KUKA KRL program: DEMO_MULTIPROC03.src, DEMO_MULTIPROC03.dat

--- DEMO_MULTIPROC03.src ---
&ACCESS RVO
&REL 23
&COMMENT MultiProc03
&PARAM DISKPATH = KRC:\R1\Program\PlcDemo
DEF  DEMO_MULTIPROC03 ( )
;********************************

;CREATOR : SPEEDBOT
;DATE    : 2024-09-23
;PROGRAM : DEMO_MULTIPROC03

;********************************
;FOLD INI;%{PE}
  ;FOLD BASISTECH INI
    GLOBAL INTERRUPT DECL 3 WHEN $STOPMESS==TRUE DO IR_STOPM ( )
    INTERRUPT ON 3
    BAS (#INITMOV,0 )
  ;ENDFOLD (BASISTECH INI)
  ;FOLD USER INI
    ;Make your modifications here
    continue
    if $MOVE_BCO == FALSE Then
      ; BCO
      ptp cur_jpos_()
    endif
  ;ENDFOLD (USER INI)
;ENDFOLD (INI)

;Example program for Process 1

;waiting for PLC clearance to proceed
;FOLD PLC.RequestToContinue ;%{PE}
req_to_continue_()
;ENDFOLD
;FOLD PLC.PathSegment IN Segment Nr: 124 ;%{PE}
path_segment_(124)
;ENDFOLD

;entering interference zone 1 with robot *.
;Enter Zone With R***
;FOLD PLC.EnterZone IN Zone Nr: ZONE [1] ;%{PE}
zone_ctrl_(#I_ENTER, 1)
;ENDFOLD

;Teach the robot to execute the first process trajectory.
;FOLD SPTP P1 CONT Vel=100 % PDAT1 Tool[1] Base[0] ;%{PE}
;FOLD Parameters ;%{h}
;Params IlfProvider=kukaroboter.basistech.inlineforms.movement.spline; Kuka.IsGlobalPoint=False; Kuka.PointName=P1; Kuka.BlendingEnabled=True; Kuka.MoveDataPtpName=PDAT1; Kuka.VelocityPtp=100; Kuka.VelocityFieldEnabled=True; Kuka.ColDetectFieldEnabled=True; Kuka.CurrentCDSetIndex=0; Kuka.MovementParameterFieldEnabled=True; IlfCommand=SPTP
;ENDFOLD
SPTP XP1 WITH $VEL_AXIS[1] = SVEL_JOINT(100.0), $TOOL = STOOL2(FP1), $BASE = SBASE(FP1.BASE_NO), $IPO_MODE = SIPO_MODE(FP1.IPO_FRAME), $LOAD = SLOAD(FP1.TOOL_NO), $ACC_AXIS[1] = SACC_JOINT(PPDAT1), $APO = SAPO_PTP(PPDAT1), $GEAR_JERK[1] = SGEAR_JERK(PPDAT1), $COLLMON_TOL_PRO[1] = USE_CM_PRO_VALUES(0) C_Spl
;ENDFOLD
;FOLD SPTP P2 CONT Vel=100 % PDAT2 Tool[1] Base[0] ;%{PE}
;FOLD Parameters ;%{h}
;Params IlfProvider=kukaroboter.basistech.inlineforms.movement.spline; Kuka.IsGlobalPoint=False; Kuka.PointName=P2; Kuka.BlendingEnabled=True; Kuka.MoveDataPtpName=PDAT2; Kuka.VelocityPtp=100; Kuka.VelocityFieldEnabled=True; Kuka.ColDetectFieldEnabled=True; Kuka.CurrentCDSetIndex=0; Kuka.MovementParameterFieldEnabled=True; IlfCommand=SPTP
;ENDFOLD
SPTP XP2 WITH $VEL_AXIS[1] = SVEL_JOINT(100.0), $TOOL = STOOL2(FP2), $BASE = SBASE(FP2.BASE_NO), $IPO_MODE = SIPO_MODE(FP2.IPO_FRAME), $LOAD = SLOAD(FP2.TOOL_NO), $ACC_AXIS[1] = SACC_JOINT(PPDAT2), $APO = SAPO_PTP(PPDAT2), $GEAR_JERK[1] = SGEAR_JERK(PPDAT2), $COLLMON_TOL_PRO[1] = USE_CM_PRO_VALUES(0) C_Spl
;ENDFOLD
;FOLD SPTP P3 CONT Vel=100 % PDAT3 Tool[1] Base[0] ;%{PE}
;FOLD Parameters ;%{h}
;Params IlfProvider=kukaroboter.basistech.inlineforms.movement.spline; Kuka.IsGlobalPoint=False; Kuka.PointName=P3; Kuka.BlendingEnabled=True; Kuka.MoveDataPtpName=PDAT3; Kuka.VelocityPtp=100; Kuka.VelocityFieldEnabled=True; Kuka.ColDetectFieldEnabled=True; Kuka.CurrentCDSetIndex=0; Kuka.MovementParameterFieldEnabled=True; IlfCommand=SPTP
;ENDFOLD
SPTP XP3 WITH $VEL_AXIS[1] = SVEL_JOINT(100.0), $TOOL = STOOL2(FP3), $BASE = SBASE(FP3.BASE_NO), $IPO_MODE = SIPO_MODE(FP3.IPO_FRAME), $LOAD = SLOAD(FP3.TOOL_NO), $ACC_AXIS[1] = SACC_JOINT(PPDAT3), $APO = SAPO_PTP(PPDAT3), $GEAR_JERK[1] = SGEAR_JERK(PPDAT3), $COLLMON_TOL_PRO[1] = USE_CM_PRO_VALUES(0) C_Spl
;ENDFOLD
;FOLD SLIN P4 CONT Vel=2 m/s CPDAT1 Tool[1] Base[0] ;%{PE}
;FOLD Parameters ;%{h}
;Params IlfProvider=kukaroboter.basistech.inlineforms.movement.spline; Kuka.IsGlobalPoint=False; Kuka.PointName=P4; Kuka.BlendingEnabled=True; Kuka.MoveDataName=CPDAT1; Kuka.VelocityPath=2; Kuka.VelocityFieldEnabled=True; Kuka.ColDetectFieldEnabled=True; Kuka.CurrentCDSetIndex=0; Kuka.MovementParameterFieldEnabled=True; IlfCommand=SLIN
;ENDFOLD
SLIN XP4 WITH $VEL = SVEL_CP(2.0, , LCPDAT1), $TOOL = STOOL2(FP4), $BASE = SBASE(FP4.BASE_NO), $IPO_MODE = SIPO_MODE(FP4.IPO_FRAME), $LOAD = SLOAD(FP4.TOOL_NO), $ACC = SACC_CP(LCPDAT1), $ORI_TYPE = SORI_TYP(LCPDAT1), $APO = SAPO(LCPDAT1), $JERK = SJERK(LCPDAT1), $COLLMON_TOL_PRO[1] = USE_CM_PRO_VALUES(0) C_Spl
;ENDFOLD
;FOLD SLIN P5 CONT Vel=2 m/s CPDAT2 Tool[1] Base[0] ;%{PE}
;FOLD Parameters ;%{h}
;Params IlfProvider=kukaroboter.basistech.inlineforms.movement.spline; Kuka.IsGlobalPoint=False; Kuka.PointName=P5; Kuka.BlendingEnabled=True; Kuka.MoveDataName=CPDAT2; Kuka.VelocityPath=2; Kuka.VelocityFieldEnabled=True; Kuka.ColDetectFieldEnabled=True; Kuka.CurrentCDSetIndex=0; Kuka.MovementParameterFieldEnabled=True; IlfCommand=SLIN
;ENDFOLD
SLIN XP5 WITH $VEL = SVEL_CP(2.0, , LCPDAT2), $TOOL = STOOL2(FP5), $BASE = SBASE(FP5.BASE_NO), $IPO_MODE = SIPO_MODE(FP5.IPO_FRAME), $LOAD = SLOAD(FP5.TOOL_NO), $ACC = SACC_CP(LCPDAT2), $ORI_TYPE = SORI_TYP(LCPDAT2), $APO = SAPO(LCPDAT2), $JERK = SJERK(LCPDAT2), $COLLMON_TOL_PRO[1] = USE_CM_PRO_VALUES(0) C_Spl
;ENDFOLD
;FOLD SLIN P6 CONT Vel=2 m/s CPDAT3 Tool[1] Base[0] ;%{PE}
;FOLD Parameters ;%{h}
;Params IlfProvider=kukaroboter.basistech.inlineforms.movement.spline; Kuka.IsGlobalPoint=False; Kuka.PointName=P6; Kuka.BlendingEnabled=True; Kuka.MoveDataName=CPDAT3; Kuka.VelocityPath=2; Kuka.VelocityFieldEnabled=True; Kuka.ColDetectFieldEnabled=True; Kuka.CurrentCDSetIndex=0; Kuka.MovementParameterFieldEnabled=True; IlfCommand=SLIN
;ENDFOLD
SLIN XP6 WITH $VEL = SVEL_CP(2.0, , LCPDAT3), $TOOL = STOOL2(FP6), $BASE = SBASE(FP6.BASE_NO), $IPO_MODE = SIPO_MODE(FP6.IPO_FRAME), $LOAD = SLOAD(FP6.TOOL_NO), $ACC = SACC_CP(LCPDAT3), $ORI_TYPE = SORI_TYP(LCPDAT3), $APO = SAPO(LCPDAT3), $JERK = SJERK(LCPDAT3), $COLLMON_TOL_PRO[1] = USE_CM_PRO_VALUES(0) C_Spl
;ENDFOLD
;FOLD SPTP P7 CONT Vel=100 % PDAT4 Tool[1] Base[0] ;%{PE}
;FOLD Parameters ;%{h}
;Params IlfProvider=kukaroboter.basistech.inlineforms.movement.spline; Kuka.IsGlobalPoint=False; Kuka.PointName=P7; Kuka.BlendingEnabled=True; Kuka.MoveDataPtpName=PDAT4; Kuka.VelocityPtp=100; Kuka.VelocityFieldEnabled=True; Kuka.ColDetectFieldEnabled=True; Kuka.CurrentCDSetIndex=0; Kuka.MovementParameterFieldEnabled=True; IlfCommand=SPTP
;ENDFOLD
SPTP XP7 WITH $VEL_AXIS[1] = SVEL_JOINT(100.0), $TOOL = STOOL2(FP7), $BASE = SBASE(FP7.BASE_NO), $IPO_MODE = SIPO_MODE(FP7.IPO_FRAME), $LOAD = SLOAD(FP7.TOOL_NO), $ACC_AXIS[1] = SACC_JOINT(PPDAT4), $APO = SAPO_PTP(PPDAT4), $GEAR_JERK[1] = SGEAR_JERK(PPDAT4), $COLLMON_TOL_PRO[1] = USE_CM_PRO_VALUES(0) C_Spl
;ENDFOLD
;FOLD SPTP P8 CONT Vel=100 % PDAT5 Tool[1] Base[0] ;%{PE}
;FOLD Parameters ;%{h}
;Params IlfProvider=kukaroboter.basistech.inlineforms.movement.spline; Kuka.IsGlobalPoint=False; Kuka.PointName=P8; Kuka.BlendingEnabled=True; Kuka.MoveDataPtpName=PDAT5; Kuka.VelocityPtp=100; Kuka.VelocityFieldEnabled=True; Kuka.ColDetectFieldEnabled=True; Kuka.CurrentCDSetIndex=0; Kuka.MovementParameterFieldEnabled=True; IlfCommand=SPTP
;ENDFOLD
SPTP XP8 WITH $VEL_AXIS[1] = SVEL_JOINT(100.0), $TOOL = STOOL2(FP8), $BASE = SBASE(FP8.BASE_NO), $IPO_MODE = SIPO_MODE(FP8.IPO_FRAME), $LOAD = SLOAD(FP8.TOOL_NO), $ACC_AXIS[1] = SACC_JOINT(PPDAT5), $APO = SAPO_PTP(PPDAT5), $GEAR_JERK[1] = SGEAR_JERK(PPDAT5), $COLLMON_TOL_PRO[1] = USE_CM_PRO_VALUES(0) C_Spl
;ENDFOLD

;This position has been fully cleared
;Does not interfere with the gripper and the corresponding robot.

;Report the completion of the first process cycle
;FOLD PLC.PathSegment IN Segment Nr: 154 ;%{PE}
path_segment_(154)
;ENDFOLD

;Exit the interference zone 1 with robot *.
;Enter Zone With R***
;FOLD PLC.ExitZone IN Zone Nr: ZONE [1] ;%{PE}
zone_ctrl_(#I_EXIT, 1)
;ENDFOLD

;waiting for PLC clearance to proceed
;FOLD PLC.RequestToContinue ;%{PE}
req_to_continue_()
;ENDFOLD
;FOLD PLC.PathSegment IN Segment Nr: 125 ;%{PE}
path_segment_(125)
;ENDFOLD

;entering interference zone 2 with robot *.
;Enter Zone With R***
;FOLD PLC.EnterZone IN Zone Nr: ZONE [2] ;%{PE}
zone_ctrl_(#I_ENTER, 2)
;ENDFOLD

;Teach the robot to execute the second process trajectory.
;FOLD SPTP P9 CONT Vel=100 % PDAT6 Tool[1] Base[0] ;%{PE}
;FOLD Parameters ;%{h}
;Params IlfProvider=kukaroboter.basistech.inlineforms.movement.spline; Kuka.IsGlobalPoint=False; Kuka.PointName=P9; Kuka.BlendingEnabled=True; Kuka.MoveDataPtpName=PDAT6; Kuka.VelocityPtp=100; Kuka.VelocityFieldEnabled=True; Kuka.ColDetectFieldEnabled=True; Kuka.CurrentCDSetIndex=0; Kuka.MovementParameterFieldEnabled=True; IlfCommand=SPTP
;ENDFOLD
SPTP XP9 WITH $VEL_AXIS[1] = SVEL_JOINT(100.0), $TOOL = STOOL2(FP9), $BASE = SBASE(FP9.BASE_NO), $IPO_MODE = SIPO_MODE(FP9.IPO_FRAME), $LOAD = SLOAD(FP9.TOOL_NO), $ACC_AXIS[1] = SACC_JOINT(PPDAT6), $APO = SAPO_PTP(PPDAT6), $GEAR_JERK[1] = SGEAR_JERK(PPDAT6), $COLLMON_TOL_PRO[1] = USE_CM_PRO_VALUES(0) C_Spl
;ENDFOLD
;FOLD SPTP P10 CONT Vel=100 % PDAT7 Tool[1] Base[0] ;%{PE}
;FOLD Parameters ;%{h}
;Params IlfProvider=kukaroboter.basistech.inlineforms.movement.spline; Kuka.IsGlobalPoint=False; Kuka.PointName=P10; Kuka.BlendingEnabled=True; Kuka.MoveDataPtpName=PDAT7; Kuka.VelocityPtp=100; Kuka.VelocityFieldEnabled=True; Kuka.ColDetectFieldEnabled=True; Kuka.CurrentCDSetIndex=0; Kuka.MovementParameterFieldEnabled=True; IlfCommand=SPTP
;ENDFOLD
SPTP XP10 WITH $VEL_AXIS[1] = SVEL_JOINT(100.0), $TOOL = STOOL2(FP10), $BASE = SBASE(FP10.BASE_NO), $IPO_MODE = SIPO_MODE(FP10.IPO_FRAME), $LOAD = SLOAD(FP10.TOOL_NO), $ACC_AXIS[1] = SACC_JOINT(PPDAT7), $APO = SAPO_PTP(PPDAT7), $GEAR_JERK[1] = SGEAR_JERK(PPDAT7), $COLLMON_TOL_PRO[1] = USE_CM_PRO_VALUES(0) C_Spl
;ENDFOLD
;FOLD SPTP P11 CONT Vel=100 % PDAT8 Tool[1] Base[0] ;%{PE}
;FOLD Parameters ;%{h}
;Params IlfProvider=kukaroboter.basistech.inlineforms.movement.spline; Kuka.IsGlobalPoint=False; Kuka.PointName=P11; Kuka.BlendingEnabled=True; Kuka.MoveDataPtpName=PDAT8; Kuka.VelocityPtp=100; Kuka.VelocityFieldEnabled=True; Kuka.ColDetectFieldEnabled=True; Kuka.CurrentCDSetIndex=0; Kuka.MovementParameterFieldEnabled=True; IlfCommand=SPTP
;ENDFOLD
SPTP XP11 WITH $VEL_AXIS[1] = SVEL_JOINT(100.0), $TOOL = STOOL2(FP11), $BASE = SBASE(FP11.BASE_NO), $IPO_MODE = SIPO_MODE(FP11.IPO_FRAME), $LOAD = SLOAD(FP11.TOOL_NO), $ACC_AXIS[1] = SACC_JOINT(PPDAT8), $APO = SAPO_PTP(PPDAT8), $GEAR_JERK[1] = SGEAR_JERK(PPDAT8), $COLLMON_TOL_PRO[1] = USE_CM_PRO_VALUES(0) C_Spl
;ENDFOLD
;FOLD SLIN P12 CONT Vel=2 m/s CPDAT4 Tool[1] Base[0] ;%{PE}
;FOLD Parameters ;%{h}
;Params IlfProvider=kukaroboter.basistech.inlineforms.movement.spline; Kuka.IsGlobalPoint=False; Kuka.PointName=P12; Kuka.BlendingEnabled=True; Kuka.MoveDataName=CPDAT4; Kuka.VelocityPath=2; Kuka.VelocityFieldEnabled=True; Kuka.ColDetectFieldEnabled=True; Kuka.CurrentCDSetIndex=0; Kuka.MovementParameterFieldEnabled=True; IlfCommand=SLIN
;ENDFOLD
SLIN XP12 WITH $VEL = SVEL_CP(2.0, , LCPDAT4), $TOOL = STOOL2(FP12), $BASE = SBASE(FP12.BASE_NO), $IPO_MODE = SIPO_MODE(FP12.IPO_FRAME), $LOAD = SLOAD(FP12.TOOL_NO), $ACC = SACC_CP(LCPDAT4), $ORI_TYPE = SORI_TYP(LCPDAT4), $APO = SAPO(LCPDAT4), $JERK = SJERK(LCPDAT4), $COLLMON_TOL_PRO[1] = USE_CM_PRO_VALUES(0) C_Spl
;ENDFOLD
;FOLD SLIN P13 CONT Vel=2 m/s CPDAT5 Tool[1] Base[0] ;%{PE}
;FOLD Parameters ;%{h}
;Params IlfProvider=kukaroboter.basistech.inlineforms.movement.spline; Kuka.IsGlobalPoint=False; Kuka.PointName=P13; Kuka.BlendingEnabled=True; Kuka.MoveDataName=CPDAT5; Kuka.VelocityPath=2; Kuka.VelocityFieldEnabled=True; Kuka.ColDetectFieldEnabled=True; Kuka.CurrentCDSetIndex=0; Kuka.MovementParameterFieldEnabled=True; IlfCommand=SLIN
;ENDFOLD
SLIN XP13 WITH $VEL = SVEL_CP(2.0, , LCPDAT5), $TOOL = STOOL2(FP13), $BASE = SBASE(FP13.BASE_NO), $IPO_MODE = SIPO_MODE(FP13.IPO_FRAME), $LOAD = SLOAD(FP13.TOOL_NO), $ACC = SACC_CP(LCPDAT5), $ORI_TYPE = SORI_TYP(LCPDAT5), $APO = SAPO(LCPDAT5), $JERK = SJERK(LCPDAT5), $COLLMON_TOL_PRO[1] = USE_CM_PRO_VALUES(0) C_Spl
;ENDFOLD
;FOLD SLIN P14 CONT Vel=2 m/s CPDAT6 Tool[1] Base[0] ;%{PE}
;FOLD Parameters ;%{h}
;Params IlfProvider=kukaroboter.basistech.inlineforms.movement.spline; Kuka.IsGlobalPoint=False; Kuka.PointName=P14; Kuka.BlendingEnabled=True; Kuka.MoveDataName=CPDAT6; Kuka.VelocityPath=2; Kuka.VelocityFieldEnabled=True; Kuka.ColDetectFieldEnabled=True; Kuka.CurrentCDSetIndex=0; Kuka.MovementParameterFieldEnabled=True; IlfCommand=SLIN
;ENDFOLD
SLIN XP14 WITH $VEL = SVEL_CP(2.0, , LCPDAT6), $TOOL = STOOL2(FP14), $BASE = SBASE(FP14.BASE_NO), $IPO_MODE = SIPO_MODE(FP14.IPO_FRAME), $LOAD = SLOAD(FP14.TOOL_NO), $ACC = SACC_CP(LCPDAT6), $ORI_TYPE = SORI_TYP(LCPDAT6), $APO = SAPO(LCPDAT6), $JERK = SJERK(LCPDAT6), $COLLMON_TOL_PRO[1] = USE_CM_PRO_VALUES(0) C_Spl
;ENDFOLD
;FOLD SPTP P15 CONT Vel=100 % PDAT9 Tool[1] Base[0] ;%{PE}
;FOLD Parameters ;%{h}
;Params IlfProvider=kukaroboter.basistech.inlineforms.movement.spline; Kuka.IsGlobalPoint=False; Kuka.PointName=P15; Kuka.BlendingEnabled=True; Kuka.MoveDataPtpName=PDAT9; Kuka.VelocityPtp=100; Kuka.VelocityFieldEnabled=True; Kuka.ColDetectFieldEnabled=True; Kuka.CurrentCDSetIndex=0; Kuka.MovementParameterFieldEnabled=True; IlfCommand=SPTP
;ENDFOLD
SPTP XP15 WITH $VEL_AXIS[1] = SVEL_JOINT(100.0), $TOOL = STOOL2(FP15), $BASE = SBASE(FP15.BASE_NO), $IPO_MODE = SIPO_MODE(FP15.IPO_FRAME), $LOAD = SLOAD(FP15.TOOL_NO), $ACC_AXIS[1] = SACC_JOINT(PPDAT9), $APO = SAPO_PTP(PPDAT9), $GEAR_JERK[1] = SGEAR_JERK(PPDAT9), $COLLMON_TOL_PRO[1] = USE_CM_PRO_VALUES(0) C_Spl
;ENDFOLD
;FOLD SPTP P16 CONT Vel=100 % PDAT10 Tool[1] Base[0] ;%{PE}
;FOLD Parameters ;%{h}
;Params IlfProvider=kukaroboter.basistech.inlineforms.movement.spline; Kuka.IsGlobalPoint=False; Kuka.PointName=P16; Kuka.BlendingEnabled=True; Kuka.MoveDataPtpName=PDAT10; Kuka.VelocityPtp=100; Kuka.VelocityFieldEnabled=True; Kuka.ColDetectFieldEnabled=True; Kuka.CurrentCDSetIndex=0; Kuka.MovementParameterFieldEnabled=True; IlfCommand=SPTP
;ENDFOLD
SPTP XP16 WITH $VEL_AXIS[1] = SVEL_JOINT(100.0), $TOOL = STOOL2(FP16), $BASE = SBASE(FP16.BASE_NO), $IPO_MODE = SIPO_MODE(FP16.IPO_FRAME), $LOAD = SLOAD(FP16.TOOL_NO), $ACC_AXIS[1] = SACC_JOINT(PPDAT10), $APO = SAPO_PTP(PPDAT10), $GEAR_JERK[1] = SGEAR_JERK(PPDAT10), $COLLMON_TOL_PRO[1] = USE_CM_PRO_VALUES(0) C_Spl
;ENDFOLD

;Report the completion of the second process cycle
;FOLD PLC.PathSegment IN Segment Nr: 155 ;%{PE}
path_segment_(155)
;ENDFOLD

;Exit the interference zone 2 with robot *.
;Enter Zone With R***
;FOLD PLC.ExitZone IN Zone Nr: ZONE [2] ;%{PE}
zone_ctrl_(#I_EXIT, 2)
;ENDFOLD
END

--- DEMO_MULTIPROC03.dat ---
&ACCESS RVO
&REL 23
&COMMENT MultiProc03
&PARAM DISKPATH = KRC:\R1\Program\PlcDemo
DEFDAT  DEMO_MULTIPROC03
;FOLD EXTERNAL DECLARATIONS;%{PE}%MKUKATPBASIS,%CEXT,%VCOMMON,%P
;FOLD BASISTECH EXT;%{PE}%MKUKATPBASIS,%CEXT,%VEXT,%P
EXT  BAS (BAS_COMMAND  :IN,REAL  :IN )
DECL INT SUCCESS
;ENDFOLD (BASISTECH EXT)
;FOLD USER EXT;%{E}%MKUKATPUSER,%CEXT,%VEXT,%P
;Make your modifications here

;ENDFOLD (USER EXT)
;ENDFOLD (EXTERNAL DECLARATIONS)
DECL E6POS XP1={X 0.00,Y 0.0,Z 0.00,A 0.0,B 0.0000,C 0.0,S 0,T 0,E1 0.0,E2 0.0,E3 0.0,E4 0.0,E5 0.0,E6 0.0}
DECL FDAT FP1={TOOL_NO 1,BASE_NO 0,IPO_FRAME #BASE,POINT2[] " "}
DECL PDAT PPDAT1={VEL 100.000,ACC 100.000,APO_DIST 500.000,APO_MODE #CDIS,GEAR_JERK 100.000,EXAX_IGN 0}
DECL MODULEPARAM_T LAST_TP_PARAMS={PARAMS[] "Kuka.VelocityFieldEnabled=True; Kuka.ColDetectFieldEnabled=True; Kuka.MovementParameterFieldEnabled=True; Kuka.IsAngleEnabled=False; Kuka.PointName=P8; Kuka.FrameData.base_no=0; Kuka.FrameData.tool_no=1; Kuka.FrameData.ipo_frame=#BASE; Kuka.isglobalpoint=False; Kuka.MoveDataPtpName=PDAT5; Kuka.MovementDataPdat.apo_mode=#CDIS; Kuka.MovementDataPdat.apo_dist=500; Kuka.MovementData.vel=100; Kuka.MovementData.acc=100; Kuka.MovementData.gear_jerk=100; Kuka.MovementData.exax_ign=0; Kuka.VelocityPtp=100; Kuka.BlendingEnabled=True; Kuka.CurrentCDSetIndex=0; Kuka.MoveDataName=CPDAT3; Kuka.MovementData.apo_fac=50; Kuka.MovementData.apo_dist=500; Kuka.MovementData.axis_acc=100; Kuka.MovementData.axis_vel=100; Kuka.MovementData.circ_typ=#BASE; Kuka.MovementData.jerk_fac=50; Kuka.MovementData.ori_typ=#VAR; Kuka.VelocityPath=2      "}
DECL E6POS XP2={X 0.00,Y 0.0,Z 0.00,A 0.0,B 0.0000,C 0.0,S 0,T 0,E1 0.0,E2 0.0,E3 0.0,E4 0.0,E5 0.0,E6 0.0}
DECL FDAT FP2={TOOL_NO 1,BASE_NO 0,IPO_FRAME #BASE,POINT2[] " "}
DECL PDAT PPDAT2={VEL 100.000,ACC 100.000,APO_DIST 500.000,APO_MODE #CDIS,GEAR_JERK 100.000,EXAX_IGN 0}
DECL E6POS XP3={X 0.00,Y 0.0,Z 0.00,A 0.0,B 0.0000,C 0.0,S 0,T 0,E1 0.0,E2 0.0,E3 0.0,E4 0.0,E5 0.0,E6 0.0}
DECL FDAT FP3={TOOL_NO 1,BASE_NO 0,IPO_FRAME #BASE,POINT2[] " "}
DECL PDAT PPDAT3={VEL 100.000,ACC 100.000,APO_DIST 500.000,APO_MODE #CDIS,GEAR_JERK 100.000,EXAX_IGN 0}
DECL E6POS XP4={X 0.00,Y 0.0,Z 0.00,A 0.0,B 0.0000,C 0.0,S 0,T 0,E1 0.0,E2 0.0,E3 0.0,E4 0.0,E5 0.0,E6 0.0}
DECL FDAT FP4={TOOL_NO 1,BASE_NO 0,IPO_FRAME #BASE,POINT2[] " "}
DECL LDAT LCPDAT1={VEL 2.00000,ACC 100.000,APO_DIST 500.000,APO_FAC 50.0000,AXIS_VEL 100.000,AXIS_ACC 100.000,ORI_TYP #VAR,CIRC_TYP #BASE,JERK_FAC 50.0000,GEAR_JERK 100.000,EXAX_IGN 0}
DECL E6POS XP5={X 0.00,Y 0.0,Z 0.00,A 0.0,B 0.0000,C 0.0,S 0,T 0,E1 0.0,E2 0.0,E3 0.0,E4 0.0,E5 0.0,E6 0.0}
DECL FDAT FP5={TOOL_NO 1,BASE_NO 0,IPO_FRAME #BASE,POINT2[] " "}
DECL LDAT LCPDAT2={VEL 2.00000,ACC 100.000,APO_DIST 500.000,APO_FAC 50.0000,AXIS_VEL 100.000,AXIS_ACC 100.000,ORI_TYP #VAR,CIRC_TYP #BASE,JERK_FAC 50.0000,GEAR_JERK 100.000,EXAX_IGN 0}
DECL E6POS XP6={X 0.00,Y 0.0,Z 0.00,A 0.0,B 0.0000,C 0.0,S 0,T 0,E1 0.0,E2 0.0,E3 0.0,E4 0.0,E5 0.0,E6 0.0}
DECL FDAT FP6={TOOL_NO 1,BASE_NO 0,IPO_FRAME #BASE,POINT2[] " "}
DECL LDAT LCPDAT3={VEL 2.00000,ACC 100.000,APO_DIST 500.000,APO_FAC 50.0000,AXIS_VEL 100.000,AXIS_ACC 100.000,ORI_TYP #VAR,CIRC_TYP #BASE,JERK_FAC 50.0000,GEAR_JERK 100.000,EXAX_IGN 0}
DECL E6POS XP7={X 0.00,Y 0.0,Z 0.00,A 0.0,B 0.0000,C 0.0,S 0,T 0,E1 0.0,E2 0.0,E3 0.0,E4 0.0,E5 0.0,E6 0.0}
DECL FDAT FP7={TOOL_NO 1,BASE_NO 0,IPO_FRAME #BASE,POINT2[] " "}
DECL PDAT PPDAT4={VEL 100.000,ACC 100.000,APO_DIST 500.000,APO_MODE #CDIS,GEAR_JERK 100.000,EXAX_IGN 0}
DECL E6POS XP8={X 0.00,Y 0.0,Z 0.00,A 0.0,B 0.0000,C 0.0,S 0,T 0,E1 0.0,E2 0.0,E3 0.0,E4 0.0,E5 0.0,E6 0.0}
DECL FDAT FP8={TOOL_NO 1,BASE_NO 0,IPO_FRAME #BASE,POINT2[] " "}
DECL PDAT PPDAT5={VEL 100.000,ACC 100.000,APO_DIST 500.000,APO_MODE #CDIS,GEAR_JERK 100.000,EXAX_IGN 0}
DECL E6POS XP9={X 0.00,Y 0.0,Z 0.00,A 0.0,B 0.0000,C 0.0,S 0,T 0,E1 0.0,E2 0.0,E3 0.0,E4 0.0,E5 0.0,E6 0.0}
DECL FDAT FP9={TOOL_NO 1,BASE_NO 0,IPO_FRAME #BASE,POINT2[] " "}
DECL PDAT PPDAT6={VEL 100.000,ACC 100.000,APO_DIST 500.000,APO_MODE #CDIS,GEAR_JERK 100.000,EXAX_IGN 0}
DECL E6POS XP10={X 0.00,Y 0.0,Z 0.00,A 0.0,B 0.0000,C 0.0,S 0,T 0,E1 0.0,E2 0.0,E3 0.0,E4 0.0,E5 0.0,E6 0.0}
DECL FDAT FP10={TOOL_NO 1,BASE_NO 0,IPO_FRAME #BASE,POINT2[] " "}
DECL PDAT PPDAT7={VEL 100.000,ACC 100.000,APO_DIST 500.000,APO_MODE #CDIS,GEAR_JERK 100.000,EXAX_IGN 0}
DECL E6POS XP11={X 0.00,Y 0.0,Z 0.00,A 0.0,B 0.0000,C 0.0,S 0,T 0,E1 0.0,E2 0.0,E3 0.0,E4 0.0,E5 0.0,E6 0.0}
DECL FDAT FP11={TOOL_NO 1,BASE_NO 0,IPO_FRAME #BASE,POINT2[] " "}
DECL PDAT PPDAT8={VEL 100.000,ACC 100.000,APO_DIST 500.000,APO_MODE #CDIS,GEAR_JERK 100.000,EXAX_IGN 0}
DECL E6POS XP12={X 0.00,Y 0.0,Z 0.00,A 0.0,B 0.0000,C 0.0,S 0,T 0,E1 0.0,E2 0.0,E3 0.0,E4 0.0,E5 0.0,E6 0.0}
DECL FDAT FP12={TOOL_NO 1,BASE_NO 0,IPO_FRAME #BASE,POINT2[] " "}
DECL LDAT LCPDAT4={VEL 2.00000,ACC 100.000,APO_DIST 500.000,APO_FAC 50.0000,AXIS_VEL 100.000,AXIS_ACC 100.000,ORI_TYP #VAR,CIRC_TYP #BASE,JERK_FAC 50.0000,GEAR_JERK 100.000,EXAX_IGN 0}
DECL E6POS XP13={X 0.00,Y 0.0,Z 0.00,A 0.0,B 0.0000,C 0.0,S 0,T 0,E1 0.0,E2 0.0,E3 0.0,E4 0.0,E5 0.0,E6 0.0}
DECL FDAT FP13={TOOL_NO 1,BASE_NO 0,IPO_FRAME #BASE,POINT2[] " "}
DECL LDAT LCPDAT5={VEL 2.00000,ACC 100.000,APO_DIST 500.000,APO_FAC 50.0000,AXIS_VEL 100.000,AXIS_ACC 100.000,ORI_TYP #VAR,CIRC_TYP #BASE,JERK_FAC 50.0000,GEAR_JERK 100.000,EXAX_IGN 0}
DECL E6POS XP14={X 0.00,Y 0.0,Z 0.00,A 0.0,B 0.0000,C 0.0,S 0,T 0,E1 0.0,E2 0.0,E3 0.0,E4 0.0,E5 0.0,E6 0.0}
DECL FDAT FP14={TOOL_NO 1,BASE_NO 0,IPO_FRAME #BASE,POINT2[] " "}
DECL LDAT LCPDAT6={VEL 2.00000,ACC 100.000,APO_DIST 500.000,APO_FAC 50.0000,AXIS_VEL 100.000,AXIS_ACC 100.000,ORI_TYP #VAR,CIRC_TYP #BASE,JERK_FAC 50.0000,GEAR_JERK 100.000,EXAX_IGN 0}
DECL E6POS XP15={X 0.00,Y 0.0,Z 0.00,A 0.0,B 0.0000,C 0.0,S 0,T 0,E1 0.0,E2 0.0,E3 0.0,E4 0.0,E5 0.0,E6 0.0}
DECL FDAT FP15={TOOL_NO 1,BASE_NO 0,IPO_FRAME #BASE,POINT2[] " "}
DECL PDAT PPDAT9={VEL 100.000,ACC 100.000,APO_DIST 500.000,APO_MODE #CDIS,GEAR_JERK 100.000,EXAX_IGN 0}
DECL E6POS XP16={X 0.00,Y 0.0,Z 0.00,A 0.0,B 0.0000,C 0.0,S 0,T 0,E1 0.0,E2 0.0,E3 0.0,E4 0.0,E5 0.0,E6 0.0}
DECL FDAT FP16={TOOL_NO 1,BASE_NO 0,IPO_FRAME #BASE,POINT2[] " "}
DECL PDAT PPDAT10={VEL 100.000,ACC 100.000,APO_DIST 500.000,APO_MODE #CDIS,GEAR_JERK 100.000,EXAX_IGN 0}
ENDDAT
